{attribute 'linkalways'}
{attribute 'no_explicit_call' := 'do not call this POU directly'}
{attribute 'enable_dynamic_creation'}
FUNCTION_BLOCK CollectionNode IMPLEMENTS I_CollectionNode
VAR
	collectableObject : I_Collectable;
	nextNode : I_CollectionNode;
END_VAR

PROPERTY PUBLIC Collectable : I_Collectable
GET
collectable := collectableObject;
END_GET
END_PROPERTY

METHOD PUBLIC Destroy
VAR_INPUT
END_VAR
__DELETE(THIS);
END_METHOD

METHOD FB_init : BOOL
VAR_INPUT
	bInitRetains : BOOL; // if TRUE, the retain variables are initialized (warm start / cold start)
	bInCopyCode : BOOL;  // if TRUE, the instance afterwards gets moved into the copy code (online change)
	Collectable : I_Collectable;
END_VAR
collectableObject := Collectable;
END_METHOD

PROPERTY PUBLIC Next : I_CollectionNode
GET
Next := nextNode;
END_GET
SET // PUBLIC
nextNode := Next;
END_SET
END_PROPERTY

END_FUNCTION_BLOCK

(* stored: Version 1.1.0.1, ProductVersion 3.1.4024.11
   POU CollectionNode: Id {ca324659-163c-423a-924a-d130bbe6c4fc}, SpecialFunc None
   Folder Constructor: Id {3159c69c-3c7c-4acd-8330-f3daff57fdc8}
   Property Collectable: Id {fcdc86e8-9e8e-4885-943e-27057e560e4e}
   Get Get: Id {31c9dd18-d3d6-44cd-a11d-f6b1fc310037}
   Method Destroy: Id {52151c94-c18b-4c21-b66f-3c84449673c0}
   Method FB_init: Id {1697923a-0fc8-4c2f-b924-4833ea034891}
   Property Next: Id {8e1ddf3a-4b70-487f-b591-2b5bcaf89b07}
   Get Get: Id {46ce132e-8357-4d98-8acf-9c947d626300}
   Set Set: Id {f2ac2e7c-d2be-4808-906e-c82174eb21b6} *)
